// TIA Portal V16 export
// export: Created 2024-12-03T15:41:46.5797116Z, ExportSetting WithReadOnly, DisplayName Totally Integrated Automation Portal, DisplayVersion V16 Update 6, DisplayName TIA Portal Version Control Interface, DisplayVersion V16 Update 2, DisplayName TIA Portal Openness, DisplayVersion V16 Update 6, DisplayName TIA Portal Teamcenter Gateway, DisplayVersion V16, DisplayName SINAMICS Startdrive Advanced, DisplayVersion V16 Update 5, DisplayName SINAMICS Startdrive G130, G150, S120, S150, SINAMICS MV, S210, DisplayVersion V16 Update 5, DisplayName SINAMICS Startdrive G110M, G120, G120C, G120D, G120P, G115D, DisplayVersion V16 Update 5, DisplayName STEP 7 Professional, DisplayVersion V16 Update 6, DisplayName STEP 7 Safety, DisplayVersion V16, DisplayName WinCC Advanced / Unified PC, DisplayVersion V16 Update 6
VAR_GLOBAL   // PLC tag table "CLOCK"
   System_Byte AT %MB0 : Byte;
   FirstScan AT %M0.0 : Bool;
   DiagStatusUpdate AT %M0.1 : Bool;
   AlwaysTRUE AT %M0.2 : Bool;
   AlwaysFALSE AT %M0.3 : Bool;
   Clock_Byte AT %MB1 : Byte;
   Clock_10Hz AT %M1.0 : Bool;
   Clock_5Hz AT %M1.1 : Bool;
   "Clock_2.5Hz" AT %M1.2 : Bool;
   Clock_2Hz AT %M1.3 : Bool;
   "Clock_1.25Hz" AT %M1.4 : Bool;
   Clock_1Hz AT %M1.5 : Bool;
   "Clock_0.625Hz" AT %M1.6 : Bool;
   "Clock_0.5Hz" AT %M1.7 : Bool;
END_VAR
VAR_GLOBAL CONSTANT   // user constants
   North : Int := 1;
   East : Int := 2;
   South : Int := 3;
   West : Int := 4;
   Up : Int := 1;
   Down : Int := -1;
   HoldPosition : Int := -1;
   ZPA_MODE : Int := 0;
   BUFFER_MODE : Int := 1;
   RUNTILLEND_MODE : Int := 2;
   IN : Int := -1;
   OUT : Int := 1;
   ZPA_TRAIN_MODE : Int := 4;
END_VAR
